PROGRAM Imperial_Metric_Switching
VAR PERSISTENT
	Pellet_Length_Displayed : REAL;
	Pellet_Length_Metric_Input : REAL;
	Pellet_Length_Imperial_Input : REAL;
END_VAR



IF GVL.Metric_Set_Bit THEN
		Pellet_Length_Displayed := Pellet_Length_Metric_Input;
		Pellet_Length_Imperial_Input := Pellet_Length_Metric_Input / 25.4;
ELSE
		Pellet_Length_Displayed := Pellet_Length_Imperial_Input;
		Pellet_Length_Metric_Input := Pellet_Length_Imperial_Input * 25.4;
END_IF

END_PROGRAM

(* stored: Version 1.1.0.1, ProductVersion 3.1.4024.12
   POU Imperial_Metric_Switching: Id {6f9d0641-37cb-4fae-bb7b-2d32027ad281}, SpecialFunc None *)
